(* PLC project Generated.project, CODESYS CODESYS V3.5 SP19 Patch 1 *)
(* stored: creationDateTime 2026-09-06T13:00:42.446289, modificationDateTime 2026-09-06T13:00:42.446289 *)

(* ======================================================================= 🪝 ST_fbWinch_Sensors — Mesures et feedbacks d'un treuil ─────────────────────────────────────────────────────────────── 🎯 Rôle : Retours physiques et mesures propres à l'instance treuil 📄 Doc métier : DOC/AF/AF_Partie-10_Fonction_Winch_v2.1.md 📤 Producteur : PRG_04_Treuils_Benne / acquisition 📥 Consommateur : FB_Winch 🔒 Structs cibles + champs conservés pour garder le garde-fou vitesse DANS FB_Winch (comportement bit-identique). Les champs MeasuredSpeedMps / MeasuredSpeedValid sont déclarés mais non consommés (usage aval). ======================================================================= *)
TYPE ST_fbWinch_Sensors : STRUCT
  CablePosM : REAL;  (* === POSITION ET RÉFÉRENCEMENT === Position actuelle du cable (m) *)
  Homed : BOOL;  (* Statut treuil reference *)
  HomingSuspect : BOOL;  (* Incertitude / doute sur le referencement *)
  ContactorsAllOff : BOOL;  (* === RETOURS CONTACTEURS === TRUE = relais sens + C1..C4 tous retombés (ex-FwdRevSpeedFeedbackOff) *)
  MeasuredSpeedMps : REAL;  (* === MESURE VITESSE === [cible] Mesure vitesse réelle (m/s) — usage aval *)
  MeasuredSpeedValid : BOOL;  (* [cible] Mesure exploitable — usage aval *)
  MeasuredSpeedBand : INT := 0;  (* [08a] Bande vitesse réelle validée (garde-fou conservé dans FB_Winch) *)
  SpeedGuardEnable : BOOL := TRUE;  (* === GARDE-FOU VITESSE (conservé) === [08a] Activation garde-fou changement de palier *)
  SpeedGuardReady : BOOL := FALSE;  (* [08a] Conditions de stabilité validées *)
END_STRUCT;
END_TYPE
